FUNCTION_BLOCK EQ_StopperArm (* Servo that places the stopper; 0..180 degrees (outer home 120, inner 1), no feedback; equipment IO: owns its IO points; commands Detach=0, MoveTo=1 *)
  (* Standard: 61499-2 *)
  (* Version 0.1, 2026-09-28, Project contributors, AAU Smart Production Lab *)
  PACKAGE stoppering;
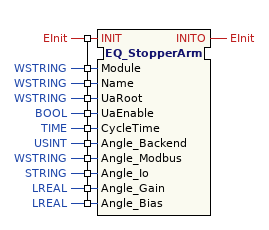
  EVENT_INPUT
    INIT : EInit WITH Module, Name, UaRoot, UaEnable, CycleTime, Angle_Backend, Angle_Modbus, Angle_Io, Angle_Gain, Angle_Bias;
  END_EVENT
  EVENT_OUTPUT
    INITO : EInit;
  END_EVENT
  VAR_INPUT
    Module : WSTRING;
    Name : WSTRING := "StopperArm";
    UaRoot : WSTRING;
    UaEnable : BOOL;
    CycleTime : TIME := T#50ms;
    Angle_Backend : USINT := 2;
    Angle_Modbus : WSTRING;
    Angle_Io : STRING;
    Angle_Gain : LREAL := 36.408;
    Angle_Bias : LREAL := 1638.4;
  END_VAR
  FBS
    Logic : stoppering::EL_StopperArm;
    Mode : modlib::MOD_StateView;
    SubCmd : iec61499::net::SUBSCRIBE_4(QI := TRUE);
    PubState : iec61499::net::PUBLISH_1(QI := TRUE);
    Out_Angle : modlib::IO_AO;
    Cycle : iec61499::events::E_CYCLE;
    PhaseT : iec61499::events::E_DELAY;
  END_FBS
  EVENT_CONNECTIONS
    INIT TO Logic.INIT;
    Logic.INITO TO Mode.INIT;
    Mode.INITO TO SubCmd.INIT;
    SubCmd.INITO TO PubState.INIT;
    PubState.INITO TO Out_Angle.INIT;
    Out_Angle.INITO TO Cycle.START;
    Out_Angle.INITO TO INITO;
    SubCmd.IND TO Logic.CMD;
    Mode.CHG TO Logic.MOD_CHG;
    Cycle.EO TO Logic.REFRESH;
    Cycle.EO TO Logic.SAMPLE;
    Logic.STATE TO PubState.REQ;
    Logic.DRIVE TO Out_Angle.REQ;
    Out_Angle.CNF TO Logic.DRIVEN;
    Logic.PHASE_START TO PhaseT.START;
    Logic.PHASE_STOP TO PhaseT.STOP;
    PhaseT.EO TO Logic.PHASE_T;
  END_CONNECTIONS
  DATA_CONNECTIONS
    Module TO Logic.Module;
    Name TO Logic.Name;
    Module TO Mode.Module;
    Logic.IdCmd TO SubCmd.ID;
    Logic.IdState TO PubState.ID;
    CycleTime TO Cycle.DT;
    SubCmd.RD_1 TO Logic.C_Holder;
    SubCmd.RD_2 TO Logic.C_Command;
    SubCmd.RD_3 TO Logic.C_Arg;
    SubCmd.RD_4 TO Logic.C_Release;
    Mode.State TO Logic.ModState;
    Logic.Holder TO PubState.SD_1;
    Angle_Backend TO Out_Angle.Backend;
    Angle_Modbus TO Out_Angle.ModbusId;
    Angle_Io TO Out_Angle.IoName;
    Logic.O_Angle TO Out_Angle.OUT;
    Logic.E_Angle TO Out_Angle.EN;
    Angle_Gain TO Out_Angle.Gain;
    Angle_Bias TO Out_Angle.Bias;
    Logic.PhaseDT TO PhaseT.DT;
  END_CONNECTIONS
END_FUNCTION_BLOCK
